(* IEC 61131-3 sources: BLM_BACKGROUND/src/PROGRAM_FILES/PROGRAMS (part 2) *)

			_PROGRAM_ENABLEAX#STATE_ENABLEAX_MODULE_0_360_TESTHEADS:
				(*{#ifdef EFLEX_DH4010}*)
					IF i_sys_first_on=TRUE THEN
						IF Modulo_0_360.outputState<>GENERAL_STATE#STATE_END THEN
							Modulo_0_360(Asse:=Y1);
						ELSE
							Modulo_0_360();
							(*{#ifdef DH4010}t*)
								CURRENT_STATE:=_PROGRAM_ENABLEAX#STATE_ENABLEAX_MODULE_0_360_TESTHEADS_2;
							(*{#else}*)
								CURRENT_STATE:=_PROGRAM_ENABLEAX#STATE_ENABLEAX_SET_STARTUP_FALSE;
							(*{#endif};*)
						END_IF;
					ELSE
						CURRENT_STATE:=_PROGRAM_ENABLEAX#STATE_ENABLEAX_SET_STARTUP_FALSE;
					END_IF;
				(*{#else}*)
					CURRENT_STATE:=_PROGRAM_ENABLEAX#STATE_ENABLEAX_SET_STARTUP_FALSE;
				(*{#endif};*)

			_PROGRAM_ENABLEAX#STATE_ENABLEAX_MODULE_0_360_TESTHEADS_2:
				(*{#ifdef DH4010}*)
					IF Modulo_0_360.outputState<>GENERAL_STATE#STATE_END THEN
						Modulo_0_360(Asse:=Y2);
					ELSE
						Modulo_0_360();
						CURRENT_STATE:=_PROGRAM_ENABLEAX#STATE_ENABLEAX_SET_STARTUP_FALSE;
					END_IF;
				(*{#endif};*)

			_PROGRAM_ENABLEAX#STATE_ENABLEAX_SET_STARTUP_FALSE:
				i_sys_ResetPressedDriver:=FALSE;
				i_sys_first_on:=FALSE;
				reset_trace(Code:=TRC_WAIT_SYSTEM_STARTUP);
				IF EnableAssi.OutputState<>GENERAL_STATE#STATE_END THEN
					EnableAssi();
				ELSE
					IF EnableAssi.ReturnValue=TRUE THEN
						CURRENT_STATE:=_PROGRAM_ENABLEAX#STATE_ENABLEAX_NUM_STATES_TEST;
					END_IF;
					EnableAssi();
				END_IF;

			_PROGRAM_ENABLEAX#STATE_ENABLEAX_NUM_STATES_TEST:
				IF TestNumStati(_Program:=PROGRAM_JOG)=FALSE THEN
					IF OPS_Active =TRUE AND OPS_StartDate=FALSE THEN
						CURRENT_STATE:=_PROGRAM_ENABLEAX#STATE_ENABLEAX_MASTER_VELOCITY_CHECK;
					ELSE
						IF i_sys_activedevice<>UNDEF_DEVICE OR i_sys_opmode<>JOGMODE THEN
							i_sys_activedevice:=UNDEF_DEVICE;
							iret:=Push_error(Code:=ERR_NUMSTATES);
						END_IF;
					END_IF;
				ELSE
					CURRENT_STATE:=_PROGRAM_ENABLEAX#STATE_ENABLEAX_MASTER_VELOCITY_CHECK;
				END_IF;

			_PROGRAM_ENABLEAX#STATE_ENABLEAX_MASTER_VELOCITY_CHECK:
				(*{#ifdef DH4010}*)
					set_trace(Code:=TRC_INCONGRUENCE_MANIPULATOR2D);
					IF disp[LOCK_2D].Enable<>Manipolatore2D_Attivo THEN
						i_sys_stopcond:=1;
					ELSE
						reset_trace(TRC_INCONGRUENCE_MANIPULATOR2D);
						IF masteraxis= AsPositioningAxisRef(Axes[X1].masteraxis) AND masteraxis^.DynamicLimits.MaxVelocity<>1 OR
							masteraxis= AsPositioningAxisRef(Axes[X2].masteraxis) AND masteraxis^.DynamicLimits.MaxVelocity<>1 THEN
						(*IF Axes[X1].masteraxis.activeconfigdata.typeofaxis.MaxVelocity.maximum<>1 OR
							 Axes[X2].masteraxis.activeconfigdata.typeofaxis.MaxVelocity.maximum<>1 THEN*)
							//Verifica che il Master abbia velocita^ 1
							dret:=Push_error(Code:=ERR_GRAVE_DOWNLOAD);
						END_IF;
						i_sys_stopcond:=0;
						i_sys_RUNOK:=1;
						CURRENT_STATE:=_PROGRAM_ENABLEAX#STATE_ENABLEAX_DEVICES_ENABLE_LOOP;
					END_IF;
				(*{#else}*)
				IF masteraxis= AsPositioningAxisRef(Axes[X1].masteraxis) AND masteraxis^.DynamicLimits.MaxVelocity<>1 THEN
					//IF Assi[X1].masteraxis.activeconfigdata.typeofaxis.MaxVelocity.maximum<>1 THEN
						//Verifica che il Master abbia velocita^ 1
						dret:=Push_error(Code:=ERR_GRAVE_DOWNLOAD);
					ELSE
						i_sys_stopcond:=0;
						i_sys_RUNOK:=1;
						(*{#ifdef MS0017}*)
							CURRENT_STATE:=_PROGRAM_ENABLEAX#STATE_ENABLEAX_HOMING_CHECK_U2;
						(*{#else}*)
							CURRENT_STATE:=_PROGRAM_ENABLEAX#STATE_ENABLEAX_DEVICES_ENABLE_LOOP;
						(*{#endif};*)
					END_IF;
				(*{#endif};*)

			_PROGRAM_ENABLEAX#STATE_ENABLEAX_HOMING_CHECK_U2:
				(*{#ifdef MS0017}*)
					PosAx:= AsPositioningAxisRef(Axes[U2].PosAx);
					IF ABS(PosAx^.actualPosition)<0.1 AND
					 	 posax^.VirtualAxis.Mode=UDINT#1 THEN
						Homing(Asse:=U2, Quota:=OldPosAxe[U2], Modo:=EnumHomingMode#DIRECT_HOMING_ABSOLUTE (*Modo:=DIRECT_HOMING*));
						CURRENT_STATE:=_PROGRAM_ENABLEAX#STATE_ENABLEAX_DEVICES_ENABLE_LOOP;
					ELSE
						CURRENT_STATE:=_PROGRAM_ENABLEAX#STATE_ENABLEAX_DEVICES_ENABLE_LOOP;
					END_IF;
				(*{#endif};*)

			_PROGRAM_ENABLEAX#STATE_ENABLEAX_DEVICES_ENABLE_LOOP:
				FOR i:=FIRST_DEVICE TO (_MAXDEVICES#MAXDEVICES+FIRST_DEVICE-1) DO
					//Disabilitazione movimento dispositivi
					AbilitazioneDispositivi(Dispositivo:=i, Stato:=TRUE);
				END_FOR;
				CURRENT_STATE:=_PROGRAM_ENABLEAX#STATE_ENABLEAX_SET_STARTUP_FALSE_FINAL;

			_PROGRAM_ENABLEAX#STATE_ENABLEAX_SET_STARTUP_FALSE_FINAL:
				i_sys_first_on:=FALSE;
				i_sys_EnableBusy:=FALSE;
				//Inizializzazione della variabile a -1 per forzare la lettura della temperatura
				//dei motori e così all^avviamento di poter attivare il feed immediatamente e non
				//attendere 1 minuto
				Appo_global :=-1;
				(*{#ifdef LINEARIZZA_ASSE} %%%%
					// FOR i:=0 TO MAX_AXIS_LINEARISES-1 DO
					// 	PosAx:=AsPositioningAxisRef(Axes[i].PosAx);
					// 	Axes[i].PosAx.servosettings.additionalcommandvalueswitch:=YES;
					// END_FOR;
				(*{#endif}	//Fine LINEARIZZA_ASSE	*)
				CURRENT_STATE:=GENERAL_STATE#STATE_END;

		 END_CASE;
		//dret:=_waitTime(T#0ms);

/*********************
 * PLC_OPEN_COMMANDS *
 *********************/
		_resetAxisError (Axis:=myPosAxis^);

		//END_WHILE;

END_PROGRAM

END_NAMESPACE

(* ---- LoadConfigurationTest.st ---- *)
USING Siemens.Simatic.S71500.Tasks;
USING Siemens.Simatic.S71500.MotionControl.Native;
USING System.BitAccess;
USING Siemens.Simatic.S71500.Clocks;
USING ENABLEPROGRAM;
USING ENABLEAX_FUNCTIONS;
USING EnableAxFunction;
USING  _TYPE;
USING Retain_Namespase;
USING _FC_FB;
USING _FC_IO_FC;
USING _CONST_VAR_DEF;
USING ENABLE_FC;

NAMESPACE _LoadConfigurationTest

PROGRAM LoadConfigurationTest

    VAR_EXTERNAL
        Axes                            		    :ARRAY[_FIRST_AXIS#FIRST_AXIS.._FIRST_AXIS#FIRST_AXIS+_CONST_VAR_DEF._MAXIS#MAXAXIS-1] OF ax;
        pm                                            : ARRAY[_FIRST_AXIS#FIRST_AXIS.._FIRST_AXIS#FIRST_AXIS+_CONST_VAR_DEF._MAXIS#MAXAXIS-1] OF AxisParameters;

        AssiMaster                      :ARRAY[FIRST_AXIS_MASTER..FIRST_AXIS_MASTER+_CONST_VAR_DEF._MAXAXIS_MASTER#MAXAXIS_MASTER-1] OF MasterAxis;
      END_VAR

      VAR_EXTERNAL CONSTANT

          FIRST_AXIS_MASTER				        :INT;

        END_VAR

////////////[AxesMaster]///////////////
      AssiMaster[0].PosAx:=UINT#200;

///////////[AxesSynchro]//////////////
      Axes[0].PosAx:=UINT#100;
      Axes[1].PosAx:=UINT#101;
      Axes[2].PosAx:=UINT#102;
      Axes[3].PosAx:=UINT#103;
      Axes[4].PosAx:=UINT#104;
      Axes[5].PosAx:=UINT#105;
      Axes[6].PosAx:=UINT#106;
      Axes[7].PosAx:=UINT#107;
      Axes[8].PosAx:=UINT#108;
      Axes[9].PosAx:=UINT#109;
      Axes[10].PosAx:=UINT#109; //!!!!!! (ifdef _maxAxsea)
      Axes[11].PosAx:=UINT#109;
      Axes[12].PosAx:=UINT#109;
      Axes[13].PosAx:=UINT#109;
      Axes[14].PosAx:=UINT#109;
      Axes[15].PosAx:=UINT#109;
      Axes[16].PosAx:=UINT#109;

      Axes[0].masteraxis:=UINT#200;
      Axes[1].masteraxis:=UINT#200;
      Axes[2].masteraxis:=UINT#200;
      Axes[3].masteraxis:=UINT#200;
      Axes[4].masteraxis:=UINT#200;
      Axes[5].masteraxis:=UINT#200;
      Axes[6].masteraxis:=UINT#200;
      Axes[7].masteraxis:=UINT#200;
      Axes[8].masteraxis:=UINT#200;
      Axes[9].masteraxis:=UINT#200;
      Axes[10].masteraxis:=UINT#200;
      Axes[11].masteraxis:=UINT#200;
      Axes[12].masteraxis:=UINT#200;
      Axes[13].masteraxis:=UINT#200;
      Axes[14].masteraxis:=UINT#200;
      Axes[15].masteraxis:=UINT#200;
      Axes[16].masteraxis:=UINT#200;

END_PROGRAM
END_NAMESPACE

(* ---- SAVE_RETAIN_PROGRAM.st ---- *)
USING Siemens.Simatic.S71500.Tasks;
USING Siemens.Simatic.S71500.MotionControl.Native;
USING Siemens.Simatic.S71500.Clocks;
USING ENABLEPROGRAM;
USING ENABLEAX_FUNCTIONS;
USING  _TYPE;
USING _FC_FB;
USING _STATE_CONST;
USING _CONST_VAR_DEF;

NAMESPACE Retain_Namespase

/**************************************************************************************
 * AT CPU SHUTDOWN, IT PERFORMS THE SAVING INTO THE RETAIN OF THE AXIS QUOTES MODULE. *
 **************************************************************************************/

// PROGRAM SaveRetain

//     VAR_EXTERNAL
// 		ProTube                     :Produzione;
// 		System_Timer                : LDATE_AND_TIME; // Timer di sistema
// 		pm                      	:ARRAY[_FIRST_AXIS#FIRST_AXIS.._FIRST_AXIS#FIRST_AXIS+_CONST_VAR_DEF._MAXIS#MAXAXIS-1] OF AxisParameters;
// 		ControlledStop				:BOOL;	//True se il Simotion è stato spento in modo controllato
// 		Axes                        :ARRAY[_FIRST_AXIS#FIRST_AXIS.._FIRST_AXIS#FIRST_AXIS+_CONST_VAR_DEF._MAXIS#MAXAXIS-1] OF ax;/// ax as structure is defined in _TYPE
// 		///ENABLEAX
// 		//ABSOLUTELY DO NOT MODIFY THE RETAIN IN THIS MODULE
// 		OldPosAxe                   :ARRAY[_FIRST_AXIS#FIRST_AXIS.._FIRST_AXIS#FIRST_AXIS+_CONST_VAR_DEF._MAXIS#MAXAXIS-1] OF LREAL;
// 		Presence4RFORM              :SINT;
// 		O_EmergencyFromSimotion		:BOOL;	//Only to be able to compile machines without safety PLCs

//     END_VAR

//     VAR_EXTERNAL CONSTANT
// 		STATE_CNC_SHUTDOWN			:INT;	//257//Gruppo 16#100 Macchina spenta;

// 		U4 							:INT;  //Mobile slide
// 		U2 							:INT;  //Core
// 		T1							:INT;	//Axis table 1
// 		T2							:INT; 	//Axis table 2
// 		A1      					:INT;  //Rotation 4RTL/"Rotazione 4RC
// 		A2      					:INT;  //Rotation 4RC
// 		B1      					:INT;  //Rotation 4RIPC
// 		B2      					:INT;  //Rotation 4RIPC
// 		V2    						:INT;  //Flow-Drill
//     END_VAR

//     VAR

// 		dret					:DINT;
// 		SettingsTO				:FB_SettingsTO;
// 		PosAx					: REF_TO TO_PositioningAxis;
// 		S_TEST : LREAL;			//TEST_LUIGI
// 	END_VAR

//     VAR_TEMP
// 		i   					:INT;
// 	END_VAR

	// ;
	// Protube.machinestate.MachineState:=STATE_CNC_SHUTDOWN; ?????-
	// Protube.machinestate.ByteHight:=SHR(TO_WORD(STATE_CNC_SHUTDOWN) & WORD#16#FF00, UINT#8);
	// Protube.machinestate.ByteLow:= TO_WORD(STATE_CNC_SHUTDOWN); //&16#00FF;
	// Protube.machinestate.datetime:=System_Timer;
	// ControlledStop:=TRUE;
	// PosAx := AsPositioningAxisRef(Axes[0].PosAx); ?????-
	// S_TEST := PosAx^.ActualPosition;//TEST_LUIGI
	// FOR i :=_FIRST_AXIS#FIRST_AXIS TO _FIRST_AXIS#FIRST_AXIS+_CONST_VAR_DEF._MAXIS#MAXAXIS-1 DO ?????-
	// 	// PosAx := AsPositioningAxisRef(Axes[0].PosAx); ?????-
	// 	IF CheckIfTOactive(Axis:=i)=TRUE THEN ;
	// 		// IF PosAx^.ActualPosition <= pm[i].Ma_Pos_Limit_Plus AND ?????-
    //         //     // PosAx^.ActualPosition >= pm[i].Ma_Pos_Limit_Minus THEN ;
	// 		// 	// //Storing axis positions only when they are not outside
	// 		// 	// //the expected limits is an attempt to avoid storing situations
	// 		// 	// //where the active positions at that time are incorrect.
	// 		// 	// OldPosAxe[0]:=PosAx^.ActualPosition; // error in TIA
	//     	// END_IF;
    // 	END_IF;
	// END_FOR;
	// (*{
	// #ifdef EMULAZIONE
	// }
	// 	{
	// 	#ifdef SMART_SMART_A
	// 	}
	// 		{
	// 		#ifdef BASCULANTE_ELETTRICO
	// 		}*)
	// 			//To enable software emulation, U4 must be enabled.
	// 			SettingsTO(Axis:=U4, State:=TRUE);
	// 			pm[U4].ma_Asse_Abilitato:=TRUE;
	// 		(*{
	// 		#endif	//Fine BASCULANTE_ELETTRICO
	// 		}
	// 	{
	// 	#endif	//Fine SMART_SMART_A
	// 	}
	// {
	// #endif	//Fine EMULAZIONE
	// }
	// {
	// #ifdef ELECTMRL
	// }
	// 	{
	// 	#ifdef TAVOLI_ELETTRICI
	// 	}*)
	// 		// SettingsTO(Axis:=T1, State:=TRUE); ?????-
	// 		// pm[T1].ma_Asse_Abilitato:=TRUE;
	// 		// SettingsTO(Axis:=T2, State:=TRUE);
	// 		// pm[T2].ma_Asse_Abilitato:=TRUE;
	// 	(*{
	// 	#endif //FINE TAVOLI_ELETTRICI
	// 	}
	// {
	// #endif //FINE ELECTMRL
	// }
	// {
	// #ifdef RUNNER
	// }*)
	// 		// This is used to ensure that BlmMotion can complete the WRITE TO CN command,
	// 		// as the TO objects of A1, B1, and B2 are destroyed when they are not enabled
	// 		// and there would be no structure to complete the data reception from BlmMotion,
	// 		// which sends the parameters in any case.
	// 		// It will be the subsequent restart of Simotion that, depending on the parameter pm[x].ma_asse_installato,
	// 		// the TO will be readjusted to the piece transferred from VGP.
	// 	// IF Presence4RFORM>0 THEN  ?????-
	// 	// 	(*{
	// 	// 	#ifndef PLAUNO_LIGHT
	// 	// 	}*)
	// 	// 		SettingsTO(Axis:=A1, State:=TRUE);
	// 	// 		pm[A1].ma_Asse_Abilitato:=TRUE;
	// 	// 		(*{
	// 	// 		#ifdef FOUR_RUNNER_PLAUNO
	// 	// 		}*)
	// 	// 			SettingsTO(Axis:=A2, State:=TRUE);
	// 	// 			pm[A2].ma_Asse_Abilitato:=TRUE;
	// 	// 		(*{
	// 	// 		#endif	//Fine FOUR_RUNNER_PLAUNO
	// 	// 		}
	// 	// 	{
	// 	// 	#endif //FINE NO PLAUNO_LIGHT
	// 	// 	}
	// 	// 	;*)
	// 	// END_IF;
	// 	(*{
	// 	#ifdef B1_B2
	// 	}*)
	// 		SettingsTO(Axis:=B1, State:=TRUE);
	// 		pm[B1].ma_Asse_Abilitato:=TRUE;
	// 		SettingsTO(Axis:=B2, State:=TRUE);
	// 		pm[B2].ma_Asse_Abilitato:=TRUE;
	// 	(*{
	// 	#endif	//Fine B1_B2
	// 	}
	// 	{
	// 	#ifdef FOUR_RUNNER
	// 	}
	// 		//The TO is reconstructed, otherwise, upon the next transition to RUN,
	// 		the error of the technological object not being closed appears. !!!!*)
	// 		SettingsTO(Axis:=V2, State:=TRUE);
	// 	(*{
	// 	#endif	//Fine FOUR_RUNNER
	// 	}
	// {
	// #endif	//Fine RUNNER
	// }
	// {
	// #ifdef PROFINET
	// }*)
	// 	O_EmergencyFromSimotion:=TRUE;
	// 	//dret:=_waitTime(T#300ms);
	// (*{
	// #endif	//Fine PROFINET
	// }*)
// END_PROGRAM
END_NAMESPACE
